TYPE ST_NC_EncDataIn :
STRUCT
	nInData1	: ARRAY[0..1] OF UINT;
	nInData2	: ARRAY[0..1] OF UINT;
	nStatus1	: BYTE;
	nStatus2	: BYTE;
	nStatus3	: BYTE;
	nStatus4	: BYTE;
END_STRUCT
END_TYPE

(* stored: Version 1.1.0.1, ProductVersion 3.1.4024.15
   DUT ST_NC_EncDataIn: Id {355f8a3d-dfc1-47ac-8c76-29a802738e48} *)
